Fanuc KAREL source: kb00073.KL

-- PROVISIONAL review KL for V940-1; original PC SHA256 760b81a6d22300d13bd3d4b2307f471da9c161061fbd4653612ceacb88e06a63
-- Incomplete behavior may be omitted. Consult companion uncertainty JSON. Do not deploy.
PROGRAM KB00073
%NOLOCKGROUP
BEGIN
  -- V9_ZERO_TABLE_METADATA_HINT layout=0002_ascii; no indexed target words; source/name/runtime held
  -- UNRESOLVED_PC offsets 5-12; opcodes 9D,23
  -- UNRESOLVED_PC offsets 17-26; opcodes 3F,75
  -- UNRESOLVED_PC offsets 31-49; opcodes 27,22,22,2A,31
  -- UNRESOLVED_PC offsets 54-58; opcodes 7F
END KB00073
